FUNCTION_BLOCK FB_ReceiptData
VAR_INPUT
	bSaveReceipt			: BOOL;
	bLoadReceipt			: BOOL;
	bDeleteReceipt			: BOOL;
	nSelectedRow			: INT;
	bHmiOk					: BOOL;
	bHmiCancel				: BOOL;
	sReceiptName			: STRING;
	sReceiptFolder			: STRING;
	pAdrrData				: PVOID;
	nLenData				: UDINT;
END_VAR
VAR_OUTPUT
	bBusy					: BOOL;
	bDone					: BOOL;
	bError					: BOOL;
	nErrorId				: UDINT;	
	sMessage				: STRING;
	aReceiptFileList		: ARRAY[0..nReceiptNum] OF STRING;
END_VAR
VAR
	(* List Receipt Files *)
	fbEnumFindFileList		: FB_EnumFindFileList;	
	stReceiptFileList		: ARRAY[0..nReceiptNum] OF ST_FindFileEntry;

	(* ReceiptList *)
	fbFileReadWrite			: FB_FileReadWrite;
	fbFileDelete			: FB_FileDelete;
	nFindReceiptListState	: INT;
	tonRefreshList			: Ton;
	nLocation				: INT;
	sFileName				: STRING(255);
	i_ReceiptFileList		: UINT;
	
	(* ReceiptState *)
	nReceiptState			: UDINT;
	bReceiptListBusy		: BOOL;
	bReceiptListDone		: BOOL;
	bReceiptListError		: BOOL;
	sFilePath				: STRING(255);
	sReceiptFileUnderOp		: STRING;
	tonMessageTimeout		: TON;
	bError_RecOp			: BOOL;
	Re_bHmiOk				: R_TRIG;
	Re_bHmiCancel			: R_TRIG;
END_VAR



(* R_TRIG --------------------------------------------------------------------------------------*)
	Re_bHmiOk(CLK:=bHmiOk);
	Re_bHmiCancel(CLK:=bHmiCancel);
(* R_TRIG --------------------------------------------------------------------------------------*)



(* FindReceiptList -----------------------------------------------------------------------------*)	
	CASE nFindReceiptListState OF
		
		0: (* Idle *)
			bReceiptListBusy:=FALSE;
			bReceiptListDone:=FALSE;
			tonRefreshList(IN:=NOT(tonRefreshList.Q) , PT:=T#3S , Q=> , ET=> );
			IF NOT(bBusy) AND tonRefreshList.Q THEN
				bReceiptListBusy:=TRUE;
				tonRefreshList(IN:=FALSE , PT:=T#3S , Q=> , ET=> );
				nFindReceiptListState:=10;
			END_IF	
			
	
		10: (* Refresh Receipt List *)
			fbEnumFindFileList(
				sNetId		:= '', 
				sPathName	:= CONCAT(sReceiptFolder,'*Backup.dat'), 
				eCmd		:= eEnumCmd_First, 
				pFindList	:= ADR(stReceiptFileList), 
				cbFindList	:= SIZEOF(stReceiptFileList), 
				bExecute	:= TRUE, 
				tTimeout	:= T#5S, 
				bBusy		=> , 
				bError		=> , 
				nErrID		=> , 
				bEOE		=> , 
				nFindFiles	=> );		
				
			IF NOT(fbEnumFindFileList.bError) THEN
				IF NOT(fbEnumFindFileList.bBusy) THEN	
					fbEnumFindFileList(
						sNetId		:= '', 
						sPathName	:= CONCAT(sReceiptFolder,'*Backup.dat'), 
						eCmd		:= eEnumCmd_First, 
						pFindList	:= ADR(stReceiptFileList), 
						cbFindList	:= SIZEOF(stReceiptFileList), 
						bExecute	:= FALSE, 
						tTimeout	:= T#5S, 
						bBusy		=> , 
						bError		=> , 
						nErrID		=> , 
						bEOE		=> , 
						nFindFiles	=> );			
					bReceiptListError:=FALSE;
					sMessage:='';
					nFindReceiptListState:=20;
				END_IF
			ELSE
				bReceiptListError:=TRUE;
				sMessage:='Receipt List could not be read';
				nFindReceiptListState:=9999;
			END_IF
		
			
		20:
			FOR i_ReceiptFileList:=0 TO nReceiptNum BY 1 DO
				nLocation:=FIND(stReceiptFileList[i_ReceiptFileList].sFileName,'Backup');
				IF nLocation<>0 THEN
					sFileName:=DELETE(stReceiptFileList[i_ReceiptFileList].sFileName,6,nLocation);
					nLocation:=FIND(sFileName,'.dat');
					aReceiptFileList[i_ReceiptFileList]:=DELETE(sFileName,4,nLocation);
				ELSE
					aReceiptFileList[i_ReceiptFileList]	:= '';
				END_IF
			END_FOR
			nFindReceiptListState:=100;
	
					
		100:
			bReceiptListDone:=TRUE;
			nFindReceiptListState:=0;
			
			
		9999:
			nFindReceiptListState:=0;

	END_CASE
(* FindReceiptList -----------------------------------------------------------------------------*)	



(* ReceiptState --------------------------------------------------------------------------------*)
	CASE nReceiptState OF
	
		0:
			bBusy:=FALSE;
			bDone:=FALSE;
			bError_RecOp:=FALSE;
			IF NOT(bReceiptListBusy OR bReceiptListError) THEN
				IF bLoadReceipt	THEN
					bBusy:=TRUE;
					nReceiptState:=100;
				ELSIF bSaveReceipt THEN
					bBusy:=TRUE;
					nReceiptState:=200;			
				ELSIF bDeleteReceipt THEN
					bBusy:=TRUE;
					nReceiptState:=300;			
				END_IF
			END_IF
				
			
		100: (* Load Receipt File *)			
			IF aReceiptFileList[nSelectedRow]<>'' THEN
				sReceiptFileUnderOp:=aReceiptFileList[nSelectedRow];
				sFilePath:=CONCAT(CONCAT(sReceiptFolder,aReceiptFileList[nSelectedRow]),'.dat');
				nReceiptState:=110;	
			ELSE
				bError_RecOp:=TRUE;
				nErrorId:=100;
				sMessage:='Receipt File is not selected';
				nReceiptState:=9999;	
			END_IF
		
			
		110: (* Loading Receipt OK / CANCEL *)
			sMessage:=CONCAT(CONCAT('Receipt : ',sReceiptFileUnderOp), ' will be loaded');	
			IF bHmiOK THEN
				nReceiptState:=120;	
			ELSIF bHmiCancel THEN
				sMessage:='Receipt Loading canceled';
				nReceiptState:=130;	
			END_IF
			
			
		120: (* Read File *)
			fbFileReadWrite(
				sFilePath		:= sFilePath, 
				bRead			:= TRUE, 
				bWrite			:= FALSE, 
				pAdrrData		:= pAdrrData, 
				nLenData		:= nLenData, 
				bBusy			=> , 
				bDone			=> , 
				bError			=> , 
				nErrorId		=> , 
				sMessage		=> , 
				tLastProcessTime=> );	
				
			IF NOT(fbFileReadWrite.bError) THEN
				IF fbFileReadWrite.bDone THEN
					fbFileReadWrite(
						sFilePath		:= sFilePath, 
						bRead			:= FALSE, 
						bWrite			:= FALSE, 
						pAdrrData		:= pAdrrData,
						nLenData		:= nLenData, 
						bBusy			=> , 
						bDone			=> , 
						bError			=> , 
						nErrorId		=> , 
						sMessage		=> , 
						tLastProcessTime=> );	
					bError_RecOp:=FALSE;
					nErrorId:=0;
					sMessage:='Receipt File is loaded';
					nReceiptState:=130;				
				END_IF
			ELSE
				bError_RecOp:=TRUE;
				nErrorId:=fbFileReadWrite.nErrorId;
				sMessage:=fbFileReadWrite.sMessage;
				nReceiptState:=9999;	
			END_IF
				
			
		130: (* Message *)
			bDone:=TRUE;
			tonMessageTimeout(IN:=TRUE , PT:=T#5S , Q=> , ET=> );
			IF NOT(bLoadReceipt) AND tonMessageTimeout.Q OR Re_bHmiOk.Q OR Re_bHmiCancel.Q THEN
				tonMessageTimeout(IN:=FALSE , PT:=T#5S , Q=> , ET=> );
				sMessage:='';
				nReceiptState:=0;		
			END_IF
		
			
		200: (* Save Receipt File *)
			IF sReceiptName<>'' THEN
				sFilePath:=CONCAT(sReceiptFolder,CONCAT(sReceiptName,'.dat'));
				sReceiptFileUnderOp:=sReceiptName;
				nReceiptState:=210;	
			ELSE
				IF aReceiptFileList[nSelectedRow]<>'' THEN
					sFilePath:=CONCAT(sReceiptFolder,CONCAT(aReceiptFileList[nSelectedRow],'.dat'));
					sReceiptFileUnderOp:=aReceiptFileList[nSelectedRow];
					sReceiptName:=aReceiptFileList[nSelectedRow];
					nReceiptState:=210;	
				ELSE	
					bError_RecOp:=TRUE;
					nErrorId:=200;
					sMessage:='Receipt File Name is not valid';
					nReceiptState:=9999;
				END_IF
			END_IF
							

		210: (* Message *)
			sMessage:=CONCAT(CONCAT('Receipt : ',sReceiptFileUnderOp), ' will be saved');	
			IF bHmiOK THEN
				nReceiptState:=220;	
			ELSIF bHmiCancel THEN
				sMessage:='Receipt Saving canceled';
				nReceiptState:=250;	
			END_IF

		
		220: (* Write File *)
			fbFileReadWrite(
				sFilePath		:= sFilePath, 
				bRead			:= FALSE, 
				bWrite			:= TRUE, 
				pAdrrData		:= pAdrrData, 
				nLenData		:= nLenData, 
				bBusy			=> , 
				bDone			=> , 
				bError			=> , 
				nErrorId		=> , 
				sMessage		=> , 
				tLastProcessTime=> );	

			IF NOT(fbFileReadWrite.bError) THEN
				IF fbFileReadWrite.bDone THEN
					fbFileReadWrite(
						sFilePath		:= sFilePath, 
						bRead			:= FALSE, 
						bWrite			:= FALSE, 
						pAdrrData		:= pAdrrData, 
						nLenData		:= nLenData, 
						bBusy			=> , 
						bDone			=> , 
						bError			=> , 
						nErrorId		=> , 
						sMessage		=> , 
						tLastProcessTime=> );		
					bError_RecOp:=FALSE;
					nErrorId:=0;	
					sMessage:='Receipt File is saved';				
					nReceiptState:=230;				
				END_IF
			ELSE
				bError_RecOp:=TRUE;
				nErrorId:=fbFileReadWrite.nErrorId;
				sMessage:=fbFileReadWrite.sMessage;
				nReceiptState:=9999;	
			END_IF
	
			
		230: (* Message *)
			IF sReceiptName<>'' THEN
				sFilePath:=CONCAT(sReceiptFolder,CONCAT(CONCAT(sReceiptName,'Backup'),'.dat'));
			ELSE
				sFilePath:=CONCAT(sReceiptFolder,CONCAT(CONCAT(aReceiptFileList[nSelectedRow],'Backup'),'.dat'));
			END_IF
			nReceiptState:=240;			
	
		
		240: (* Write Backup File *)
			fbFileReadWrite(
				sFilePath		:= sFilePath, 
				bRead			:= FALSE, 
				bWrite			:= TRUE, 
				pAdrrData		:= pAdrrData, 
				nLenData		:= nLenData, 
				bBusy			=> , 
				bDone			=> , 
				bError			=> , 
				nErrorId		=> , 
				sMessage		=> , 
				tLastProcessTime=> );	

			IF NOT(fbFileReadWrite.bError) THEN
				IF fbFileReadWrite.bDone THEN
					fbFileReadWrite(
						sFilePath		:= sFilePath, 
						bRead			:= FALSE, 
						bWrite			:= FALSE, 
						pAdrrData		:= pAdrrData, 
						nLenData		:= nLenData, 
						bBusy			=> , 
						bDone			=> , 
						bError			=> , 
						nErrorId		=> , 
						sMessage		=> , 
						tLastProcessTime=> );					
					bError_RecOp:=FALSE;
					nErrorId:=0;		
					sMessage:='Receipt File is saved'; (* Receipt and Backup Files are saved *)
					nReceiptState:=250;				
				END_IF
			ELSE
				bError_RecOp:=TRUE;
				nErrorId:=fbFileReadWrite.nErrorId;
				sMessage:=fbFileReadWrite.sMessage;
				nReceiptState:=9999;	
			END_IF	
				
				
		250: (* Message *)
			bDone:=TRUE;
			tonMessageTimeout(IN:=TRUE , PT:=T#5S , Q=> , ET=> );
			IF NOT(bSaveReceipt) AND tonMessageTimeout.Q OR Re_bHmiOk.Q OR Re_bHmiCancel.Q  THEN
				tonMessageTimeout(IN:=FALSE , PT:=T#5S , Q=> , ET=> );
				sMessage:='';
				nReceiptState:=0;		
			END_IF			
		
			
		300: (* Delete Receipt File *)					
			IF aReceiptFileList[nSelectedRow]<>'' THEN
				sReceiptFileUnderOp:=aReceiptFileList[nSelectedRow];
				sFilePath:=CONCAT(CONCAT(sReceiptFolder,aReceiptFileList[nSelectedRow]),'.dat');
				nReceiptState:=310;	
			ELSE
				bError_RecOp:=TRUE;
				nErrorId:=300;
				sMessage:='Receipt File is not selected';
				nReceiptState:=9999;	
			END_IF			
			
			
		310: (* Message *)
			sMessage:=CONCAT(CONCAT('Receipt : ',sReceiptFileUnderOp), ' will be deleted');	
			IF bHmiOK THEN
				nReceiptState:=320;	
			ELSIF bHmiCancel THEN
				sMessage:='Receipt Deleting canceled';
				nReceiptState:=350;	
			END_IF	
					
			
		320: (* Delete Receipt File *)
			fbFileDelete(
				sNetId		:= '', 
				sPathName	:= sFilePath, 
				ePath		:= , 
				bExecute	:= TRUE, 
				tTimeout	:= , 
				bBusy		=> , 
				bError		=> , 
				nErrId		=> );
			
			IF NOT(fbFileDelete.bError) THEN
				IF NOT(fbFileDelete.bBusy) THEN
					fbFileDelete(
						sNetId		:= '', 
						sPathName	:= sFilePath, 
						ePath		:= , 
						bExecute	:= FALSE, 
						tTimeout	:= , 
						bBusy		=> , 
						bError		=> , 
						nErrId		=> );	
					bError_RecOp:=FALSE;
					nErrorId:=0;
					sMessage:='Receipt File is deleted';
					nReceiptState:=330;	
				END_IF
			ELSE
				bError_RecOp:=TRUE;
				nErrorId:=fbFileDelete.nErrId;
				sMessage:='Receipt File Deleting Error';
				nReceiptState:=9999;
			END_IF
			
			
		330: (* Message *)		
			sFilePath:=CONCAT(CONCAT(sReceiptFolder,CONCAT(aReceiptFileList[nSelectedRow],'Backup')),'.dat');	
			nReceiptState:=340;	
	
			
		340: (* Delete Backup File *)	
			fbFileDelete(
				sNetId		:= '', 
				sPathName	:= sFilePath, 
				ePath		:= , 
				bExecute	:= TRUE, 
				tTimeout	:= , 
				bBusy		=> , 
				bError		=> , 
				nErrId		=> );
			
			IF NOT(fbFileDelete.bError) THEN
				IF NOT(fbFileDelete.bBusy) THEN
					fbFileDelete(
						sNetId		:= '', 
						sPathName	:= sFilePath, 
						ePath		:= , 
						bExecute	:= FALSE, 
						tTimeout	:= , 
						bBusy		=> , 
						bError		=> , 
						nErrId		=> );	
					bError_RecOp:=FALSE;
					nErrorId:=0;
					sMessage:='Receipt File is deleted';	(* Receipt and Backup Files are deleted *)
					nReceiptState:=350;	
				END_IF
			ELSE
				bError_RecOp:=TRUE;
				nErrorId:=fbFileDelete.nErrId;
				sMessage:='Receipt Backup File Deleting Error';
				nReceiptState:=9999;
			END_IF
		
				
		350: (* Message *)
			bDone:=TRUE;
			tonMessageTimeout(IN:=TRUE , PT:=T#5S , Q=> , ET=> );
			IF NOT(bDeleteReceipt) AND tonMessageTimeout.Q OR Re_bHmiOk.Q OR Re_bHmiCancel.Q  THEN
				tonMessageTimeout(IN:=FALSE , PT:=T#5S , Q=> , ET=> );
				sMessage:='';
				nReceiptState:=0;		
			END_IF			

		
					
		9999:(* Error *)
			fbFileReadWrite(
				sFilePath		:= sFilePath, 
				bRead			:= FALSE, 
				bWrite			:= FALSE, 
				pAdrrData		:= pAdrrData, 
				nLenData		:= nLenData, 
				bBusy			=> , 
				bDone			=> , 
				bError			=> , 
				nErrorId		=> , 
				sMessage		=> , 
				tLastProcessTime=> );	
				
			fbFileDelete(
				sNetId		:= '', 
				sPathName	:= sFilePath, 
				ePath		:= , 
				bExecute	:= FALSE, 
				tTimeout	:= , 
				bBusy		=> , 
				bError		=> , 
				nErrId		=> );		
		
			tonMessageTimeout(IN:=TRUE , PT:=T#5S , Q=> , ET=> );			
				
			IF	NOT(fbFileReadWrite.bBusy OR fbFileDelete.bBusy)
				AND NOT(bSaveReceipt OR bLoadReceipt OR bDeleteReceipt) 
				AND (tonMessageTimeout.Q OR bHmiOK OR bHmiCancel)
			THEN
				tonMessageTimeout(IN:=FALSE , PT:=T#5S , Q=> , ET=> );		
				sMessage:='';	
				nReceiptState:=0;		
			END_IF				
	
	END_CASE
(* ReceiptState --------------------------------------------------------------------------------*)	



(* Error ---------------------------------------------------------------------------------------*)
	bError	:= (bError_RecOp OR bReceiptListError);
(* Error ---------------------------------------------------------------------------------------*)

END_FUNCTION_BLOCK

(* stored: Version 1.1.0.1, ProductVersion 3.1.4024.6
   POU FB_ReceiptData: Id {bd549986-4a1b-42c0-a973-ba67529b4aa7}, SpecialFunc None *)
